FUNCTION TryConvert_BYTE_TO_TIME : BOOL
VAR_INPUT
	in : BYTE;
	out : REFERENCE TO TIME;
END_VAR

out := BYTE_TO_TIME(in);
TryConvert_BYTE_TO_TIME := TRUE;

END_FUNCTION

(* stored: Version 1.1.0.1, ProductVersion 3.1.4024.12
   POU TryConvert_BYTE_TO_TIME: Id {9a71432d-3aaa-499c-9ce0-f7ed3535f44f}, SpecialFunc None *)
